Staubli VAL3: replacePattern.pgx

public program replacePattern(string& x_sInput[], string x_sPattern, string x_sReplace, string& x_sResult[])
  local num l_nLength
  local num l_nElement
  local string l_sText
begin

  l_nLength = size(x_sInput)
  resize(x_sResult,1,1)
  x_sResult = ""
  resize(x_sResult,1,l_nLength)

  for l_nElement = 0 to l_nLength-1
    l_sText = x_sInput[l_nElement]
    while find(l_sText,x_sPattern)!=-1
      l_sText = replace(l_sText,x_sReplace,len(x_sPattern),find(l_sText,x_sPattern))
    endWhile
    x_sResult[l_nElement] = l_sText
  endFor

end
